{attribute 'qualified_only'}
{attribute 'strict'}
TYPE SafeState :
(
	Init		:= 0,
	Close		:= 1,
	CeckDigit	:= 2,
	WrongCode	:= 3,
	Open		:= 4
	
);
END_TYPE

(* stored: Version 1.1.0.1, ProductVersion 3.1.4022.12
   DUT SafeState: Id {f5a5603a-4486-4875-bdb4-012913d9cd23} *)
